// TIA Portal V16 export
// export: Created 2021-07-12T14:47:19.537172Z, ExportSetting WithDefaults, DisplayName Totally Integrated Automation Portal, DisplayVersion V16, DisplayName TIA Portal Version Control Interface, DisplayVersion V16, DisplayName TIA Portal Openness, DisplayVersion V16, DisplayName STEP 7 Professional, DisplayVersion V16, DisplayName STEP 7 Safety, DisplayVersion V16, DisplayName WinCC Professional, DisplayVersion V16
TYPE "LSimaHydTO_typeActor"
TITLE = LSimaHydTO_typeActor
// Actor configuration
// stored: IsFailsafeCompliant false
   STRUCT
      InverseDirection { S7_SetPoint := 'True'} : Bool := FALSE;   // Inversion of the setpoint if TRUE
      BiDirectional { S7_SetPoint := 'True'} : Bool := TRUE;   // Positive and negative outputs
      SubstituteValue { S7_SetPoint := 'True'} : LReal := 0.0;   // Substitute Output Value if disabled
      MaxDerivative { S7_SetPoint := 'True'} : LReal := 10000.0;   // Limit of changes at the manipulated variable
      DirectionValves { S7_SetPoint := 'True'} : "LSimaHydTO_typeActorDirectionValves";
   END_STRUCT;
END_TYPE
